// TIA Portal V17 export
// export: Created 2026-05-13T16:54:42.1553591Z, ExportSetting WithDefaults, DisplayName Totally Integrated Automation Portal, DisplayVersion V17 Update 4, DisplayName TIA Portal Openness, DisplayVersion V17 Update 4, DisplayName TIA Portal Version Control Interface, DisplayVersion V17, DisplayName SINAMICS Startdrive Advanced, DisplayVersion V17, DisplayName SINAMICS Startdrive G130, G150, S120, S150, SINAMICS MV, S210, DisplayVersion V17, DisplayName SINAMICS Startdrive G110M, G120, G120C, G120D, G120P, G115D, DisplayVersion V17, DisplayName STEP 7 Professional, DisplayVersion V17 Update 4, DisplayName STEP 7 Safety, DisplayVersion V17, DisplayName WinCC Professional, DisplayVersion V17 Update 4
TagTable "配方"
  FB_配方_DB_当前配方_编号 : Int  (PLC tag FB_配方_DB.当前配方.编号, HMI_连接_1, 1 s)
  FB_配方_DB_当前配方_配方 : UDT_配方  (PLC tag FB_配方_DB.当前配方.配方, HMI_连接_1, 1 s)
    TagStructureMember "名称"
    TagStructureMember "JF进风温度"
    TagStructureMember "RS热水炉温度"
    TagStructureMember "HW恒温系统温度"
    TagStructureMember "JL进料泵设定"
    TagStructureMember "YF引风频率"
    TagStructureMember "LX离心雾化"
  FB_配方_DB_编辑配方_编号 : Int  (PLC tag FB_配方_DB.编辑配方.编号, HMI_连接_1, 1 s)
  FB_配方_DB_编辑配方_增加 : Bool  (PLC tag FB_配方_DB.编辑配方.增加, HMI_连接_1, 1 s)
  FB_配方_DB_编辑配方_删除 : Bool  (PLC tag FB_配方_DB.编辑配方.删除, HMI_连接_1, 1 s)
  FB_配方_DB_编辑配方_修改 : Bool  (PLC tag FB_配方_DB.编辑配方.修改, HMI_连接_1, 1 s)
  FB_配方_DB_编辑配方_修改_确认 : Bool  (PLC tag FB_配方_DB.编辑配方.修改_确认, HMI_连接_1, 1 s)
  FB_配方_DB_编辑配方_修改_取消 : Bool  (PLC tag FB_配方_DB.编辑配方.修改_取消, HMI_连接_1, 1 s)
  FB_配方_DB_编辑配方_复制 : Bool  (PLC tag FB_配方_DB.编辑配方.复制, HMI_连接_1, 1 s)
  FB_配方_DB_编辑配方_粘贴 : Bool  (PLC tag FB_配方_DB.编辑配方.粘贴, HMI_连接_1, 1 s)
  FB_配方_DB_编辑配方_应用配方 : Bool  (PLC tag FB_配方_DB.编辑配方.应用配方, HMI_连接_1, 1 s)
  FB_配方_DB_编辑配方_已复制 : Bool  (PLC tag FB_配方_DB.编辑配方.已复制, HMI_连接_1, 1 s)
  FB_配方_DB_编辑配方_记录 : Bool  (PLC tag FB_配方_DB.编辑配方.记录, HMI_连接_1, 1 s)
  FB_配方_DB_编辑配方_编辑配方 : UDT_配方  (PLC tag FB_配方_DB.编辑配方.编辑配方, HMI_连接_1, 1 s)
    TagStructureMember "名称"
    TagStructureMember "JF进风温度"
    TagStructureMember "RS热水炉温度"
    TagStructureMember "HW恒温系统温度"
    TagStructureMember "JL进料泵设定"
    TagStructureMember "YF引风频率"
    TagStructureMember "LX离心雾化"
  FB_配方_DB_编辑配方_复制配方 : UDT_配方  (PLC tag FB_配方_DB.编辑配方.复制配方, HMI_连接_1, 1 s)
    TagStructureMember "名称"
    TagStructureMember "JF进风温度"
    TagStructureMember "RS热水炉温度"
    TagStructureMember "HW恒温系统温度"
    TagStructureMember "JL进料泵设定"
    TagStructureMember "YF引风频率"
    TagStructureMember "LX离心雾化"
  FB_配方_DB_配方列表{1} : UDT_配方  (PLC tag FB_配方_DB.配方列表[1], HMI_连接_1, 1 s)
    TagStructureMember "名称"
    TagStructureMember "JF进风温度"
    TagStructureMember "RS热水炉温度"
    TagStructureMember "HW恒温系统温度"
    TagStructureMember "JL进料泵设定"
    TagStructureMember "YF引风频率"
    TagStructureMember "LX离心雾化"
  FB_配方_DB_配方列表{2} : UDT_配方  (PLC tag FB_配方_DB.配方列表[2], HMI_连接_1, 1 s)
    TagStructureMember "名称"
    TagStructureMember "JF进风温度"
    TagStructureMember "RS热水炉温度"
    TagStructureMember "HW恒温系统温度"
    TagStructureMember "JL进料泵设定"
    TagStructureMember "YF引风频率"
    TagStructureMember "LX离心雾化"
  FB_配方_DB_配方列表{3} : UDT_配方  (PLC tag FB_配方_DB.配方列表[3], HMI_连接_1, 1 s)
    TagStructureMember "名称"
    TagStructureMember "JF进风温度"
    TagStructureMember "RS热水炉温度"
    TagStructureMember "HW恒温系统温度"
    TagStructureMember "JL进料泵设定"
    TagStructureMember "YF引风频率"
    TagStructureMember "LX离心雾化"
  FB_配方_DB_配方列表{4} : UDT_配方  (PLC tag FB_配方_DB.配方列表[4], HMI_连接_1, 1 s)
    TagStructureMember "名称"
    TagStructureMember "JF进风温度"
    TagStructureMember "RS热水炉温度"
    TagStructureMember "HW恒温系统温度"
    TagStructureMember "JL进料泵设定"
    TagStructureMember "YF引风频率"
    TagStructureMember "LX离心雾化"
  FB_配方_DB_配方列表{5} : UDT_配方  (PLC tag FB_配方_DB.配方列表[5], HMI_连接_1, 1 s)
    TagStructureMember "名称"
    TagStructureMember "JF进风温度"
    TagStructureMember "RS热水炉温度"
    TagStructureMember "HW恒温系统温度"
    TagStructureMember "JL进料泵设定"
    TagStructureMember "YF引风频率"
    TagStructureMember "LX离心雾化"
  FB_配方_DB_配方列表{6} : UDT_配方  (PLC tag FB_配方_DB.配方列表[6], HMI_连接_1, 1 s)
    TagStructureMember "名称"
    TagStructureMember "JF进风温度"
    TagStructureMember "RS热水炉温度"
    TagStructureMember "HW恒温系统温度"
    TagStructureMember "JL进料泵设定"
    TagStructureMember "YF引风频率"
    TagStructureMember "LX离心雾化"
  FB_配方_DB_配方列表{7} : UDT_配方  (PLC tag FB_配方_DB.配方列表[7], HMI_连接_1, 1 s)
    TagStructureMember "名称"
    TagStructureMember "JF进风温度"
    TagStructureMember "RS热水炉温度"
    TagStructureMember "HW恒温系统温度"
    TagStructureMember "JL进料泵设定"
    TagStructureMember "YF引风频率"
    TagStructureMember "LX离心雾化"
  FB_配方_DB_配方列表{8} : UDT_配方  (PLC tag FB_配方_DB.配方列表[8], HMI_连接_1, 1 s)
    TagStructureMember "名称"
    TagStructureMember "JF进风温度"
    TagStructureMember "RS热水炉温度"
    TagStructureMember "HW恒温系统温度"
    TagStructureMember "JL进料泵设定"
    TagStructureMember "YF引风频率"
    TagStructureMember "LX离心雾化"
  FB_配方_DB_配方列表{9} : UDT_配方  (PLC tag FB_配方_DB.配方列表[9], HMI_连接_1, 1 s)
    TagStructureMember "名称"
    TagStructureMember "JF进风温度"
    TagStructureMember "RS热水炉温度"
    TagStructureMember "HW恒温系统温度"
    TagStructureMember "JL进料泵设定"
    TagStructureMember "YF引风频率"
    TagStructureMember "LX离心雾化"
  FB_配方_DB_配方列表{10} : UDT_配方  (PLC tag FB_配方_DB.配方列表[10], HMI_连接_1, 1 s)
    TagStructureMember "名称"
    TagStructureMember "JF进风温度"
    TagStructureMember "RS热水炉温度"
    TagStructureMember "HW恒温系统温度"
    TagStructureMember "JL进料泵设定"
    TagStructureMember "YF引风频率"
    TagStructureMember "LX离心雾化"
